{attribute 'qualified_only'}
{attribute 'strict'}
TYPE E_Step :
(
	// Special steps
	NoStep := -32767,	// No step
	Unknown := -32000,	// Unknown step
	
	// Not Enabled or Errors
	NeOrError := -990,	// Not enabled or at fault //
	
	// Recovery
	Recovering := 990,	// Restore After Failure //

	// Stopping
	Stopping := 900,	// Nominal shutdown //
	
	// Stop
	Stop := 0, 			// S0 Stop //
	
	// Working steps
	RecoverPunch := 50,		// S1 Lift the punch at restart //
	WaitObject := 100,		// S2 Waiting for object //
	DelayToFeeding := 120,	// S3 delay before feeding  //
	Loading := 200,			// S4 Object Transfer //
	LowerPunch := 300,		// S5 Lower the punch //
	LiftPunch := 400,		// S6 Lift the punch //
	Unloading := 500,		// S7 Outgoing object discharge //
	DelayOnUnloading := 520	// S8 delay after unloading //
   
);
END_TYPE
//  NoStep = '-32767'
//  Unknown = '-32000'
//  NeOrError = '-990'

(* stored: Version 1.1.0.1, ProductVersion 3.1.4024.12
   EnumerationTextList E_Step: Id {0845bbf6-d79e-46f5-b33c-353400a4e494} *)
